FUNCTION_BLOCK FB_Alarm EXTENDS FB_TcAlarm

VAR_INPUT
	evtEntry	: TcEventEntry;
	bEvt		: BOOL;
	bConfirm	: BOOL;
END_VAR

VAR_OUTPUT
END_VAR

VAR
	bInit  		: BOOL := TRUE;
	bMem		: BOOL;
END_VAR

IF bInit THEN
	SUPER^.CreateEx(evtEntry, TRUE, 0);
	bInit := FALSE;
END_IF

IF bEvt AND NOT bMem AND SUPER^.eConfirmationState <> TcEventConfirmationState.WaitForConfirmation THEN
	SUPER^.Raise(0);
END_IF

IF bMem AND NOT bEvt THEN
	SUPER^.Clear(0, FALSE);
END_IF

IF bConfirm THEN
	SUPER^.Confirm(0);
END_IF

bMem := bEvt;

END_FUNCTION_BLOCK

(* stored: Version 1.1.0.1, ProductVersion 3.1.4024.9
   POU FB_Alarm: Id {3e954f32-19db-46f0-a3f1-49f553186a71}, SpecialFunc None *)
